INTERFACE I_TaskCyclicEvent EXTENDS I_Event

PROPERTY Info : PlcTaskSystemInfo
GET
END_GET
END_PROPERTY

END_INTERFACE

(* stored: Version 1.1.0.1, ProductVersion 3.1.4024.11
   Itf I_TaskCyclicEvent: Id {33d43389-6006-4cda-baca-66ee2d21f4d2}
   Property Info: Id {61a79a24-7897-4fd8-8ab2-0fac4e32b5ca}
   Get Get: Id {bda09813-983c-4f63-9dfd-15c54d4fa712} *)
